% RSLogix 500 project 2 WAY TRAFFIC LIGHT 2 SENSOR_BAK001.RSS, saved by version 8.30.00.16 %
PROJECT "UNTITLED"    % processor: MicroLogix 1000 %

PROGRAM FILES
  LAD 2 "MAIN_PROG"  11 rungs
  LAD 3 "USER_FAULT"  1 rungs
  LAD 4 "HSC_INT"  1 rungs
  LAD 5 "STI_INT"  1 rungs
  LAD 6, 7, 8, 9, 10, 11, 12, 13, 14, 15, 16: only END

DATA FILES
  O0 OUTPUT  1 elements
  I1 INPUT  2 elements
  S2 STATUS  33 elements
  B3 BINARY  32 elements
  T4 TIMER  40 elements
  C5 COUNTER  32 elements
  R6 CONTROL  16 elements
  N7 INTEGER  105 elements

LADDER 2 "MAIN_PROG"
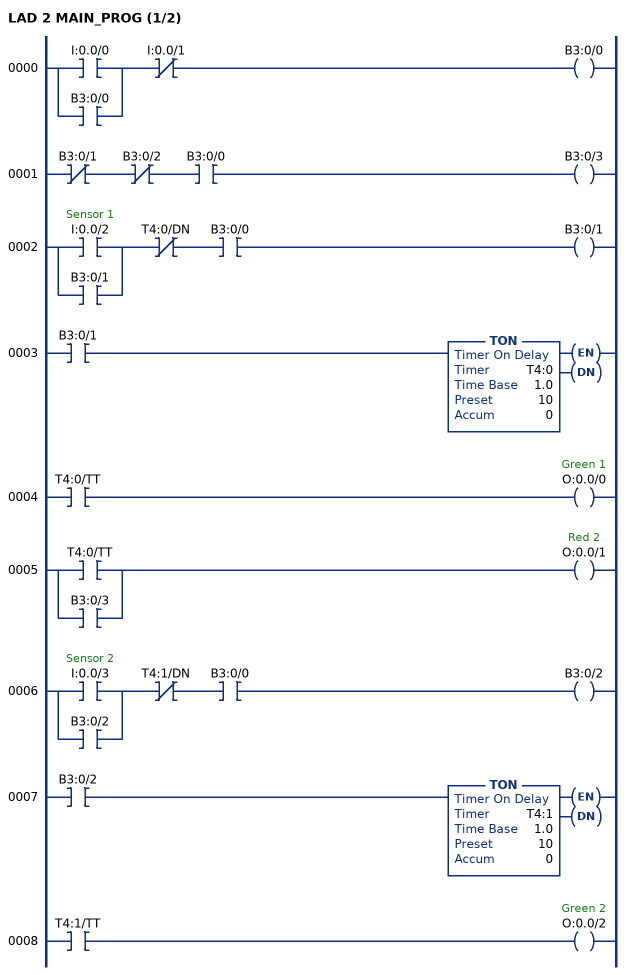
% Rung: 0 %
SOR BST XIC I:0.0/0 NXB XIC B3:0/0 BND XIO I:0.0/1 OTE B3:0/0 EOR
% Rung: 1 %
SOR XIO B3:0/1 XIO B3:0/2 XIC B3:0/0 OTE B3:0/3 EOR
% Rung: 2 %
SOR BST XIC I:0.0/2 NXB XIC B3:0/1 BND XIO T4:0/DN XIC B3:0/0 OTE B3:0/1 EOR
%   I:0.0/2  "Sensor 1" %
% Rung: 3 %
SOR XIC B3:0/1 TON T4:0 1.0 10 0 EOR
% Rung: 4 %
SOR XIC T4:0/TT OTE O:0.0/0 EOR
%   O:0.0/0  "Green 1" %
% Rung: 5 %
SOR BST XIC T4:0/TT NXB XIC B3:0/3 BND OTE O:0.0/1 EOR
%   O:0.0/1  "Red 2" %
% Rung: 6 %
SOR BST XIC I:0.0/3 NXB XIC B3:0/2 BND XIO T4:1/DN XIC B3:0/0 OTE B3:0/2 EOR
%   I:0.0/3  "Sensor 2" %
% Rung: 7 %
SOR XIC B3:0/2 TON T4:1 1.0 10 0 EOR
% Rung: 8 %
SOR XIC T4:1/TT OTE O:0.0/2 EOR
%   O:0.0/2  "Green 2" %

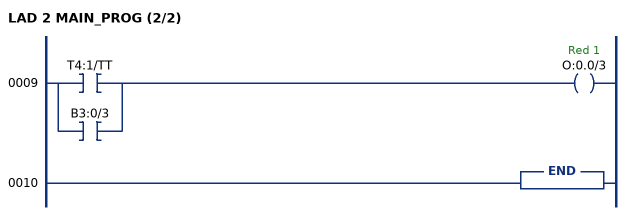
% Rung: 9 %
SOR BST XIC T4:1/TT NXB XIC B3:0/3 BND OTE O:0.0/3 EOR
%   O:0.0/3  "Red 1" %
% Rung: 10 %
SOR END EOR

DATA TABLE (non-zero values as saved)
DATA T4
% .PRE .ACC %
% T4:0 % 10 0
% T4:1 % 10 0
